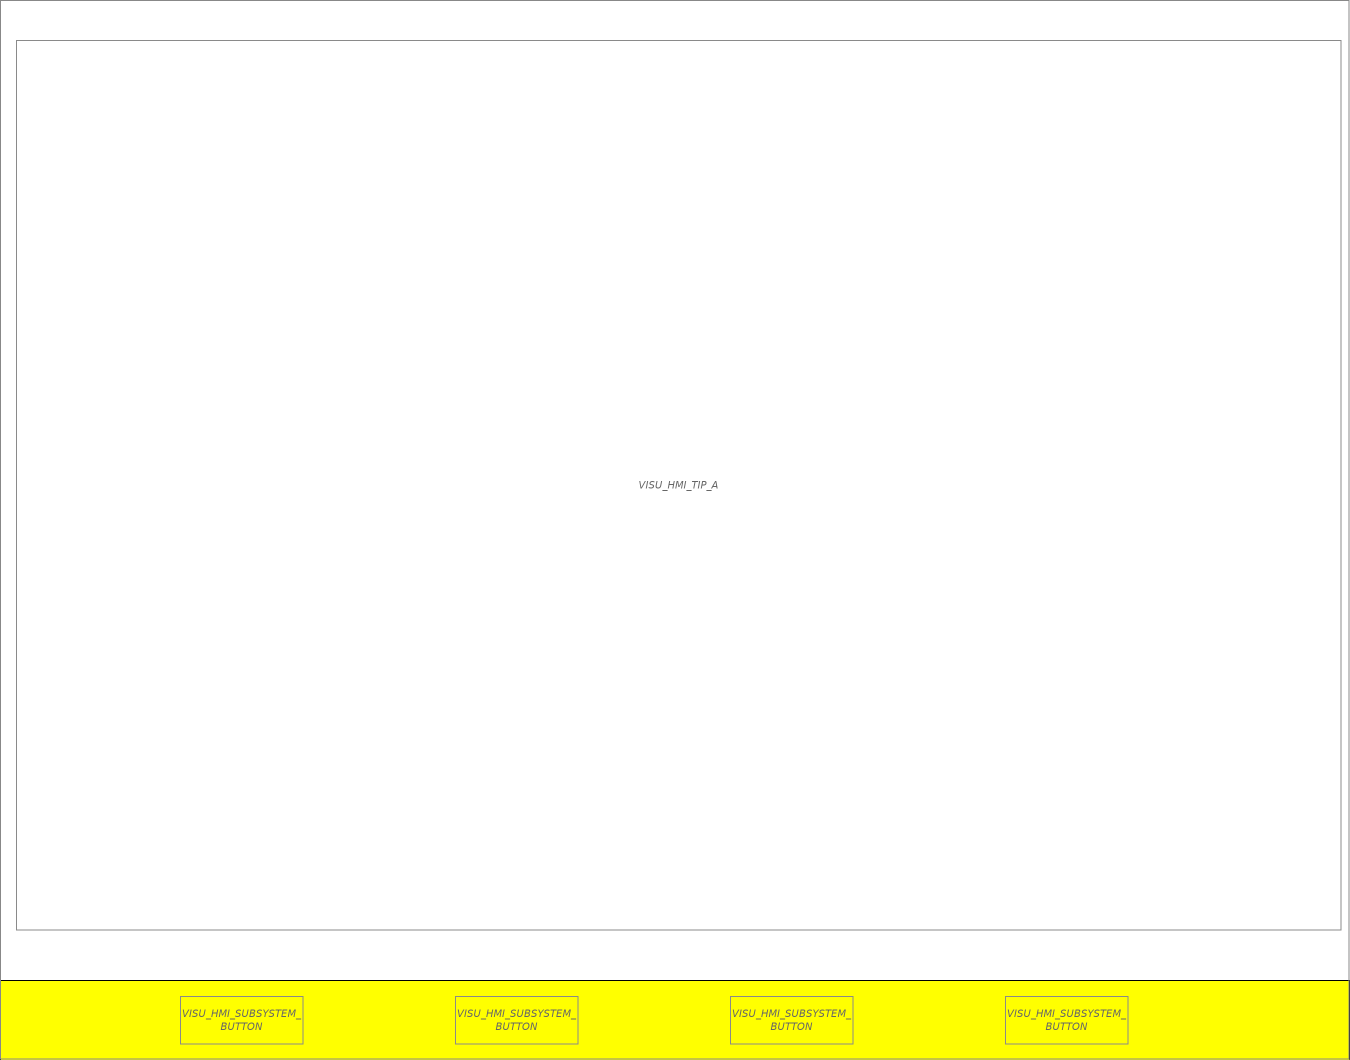
VISUALIZATION VISU_HMI_TIP_TILT  // 1350x1060
VAR_IN_OUT
	m_Hmi : FB_HMI_TIP_TILT;
END_VAR
    Label (10,10 199x30), "Tip Tilt"
    Rectangle (0,980 1350x81)
    Frame (180,996 123x48)
        shows VISU_HMI_SUBSYSTEM_BUTTON(m_Hmi := PRG_HMI.fbTipTilt.fbTipAButton)
        OnMouseClick: execute { m_Hmi.eActiveTab := E_HMI_TIP_TILT_TABS.TIP_A; }
    Frame (455,996 123x48)
        shows VISU_HMI_SUBSYSTEM_BUTTON(m_Hmi := PRG_HMI.fbTipTilt.fbTipBButton)
        OnMouseClick: execute { m_Hmi.eActiveTab := E_HMI_TIP_TILT_TABS.TIP_B; }
    Frame (730,996 123x48)
        shows VISU_HMI_SUBSYSTEM_BUTTON(m_Hmi := PRG_HMI.fbTipTilt.fbTiltAButton)
        OnMouseClick: execute { m_Hmi.eActiveTab := E_HMI_TIP_TILT_TABS.TILT_A; }
    Frame (1005,996 123x48)
        shows VISU_HMI_SUBSYSTEM_BUTTON(m_Hmi := PRG_HMI.fbTipTilt.fbTiltBButton)
        OnMouseClick: execute { m_Hmi.eActiveTab := E_HMI_TIP_TILT_TABS.TILT_B; }
    Frame (16,40 1325x890), frame switch variable: m_Hmi.eActiveTab
        shows VISU_HMI_TIP_A()
        shows VISU_HMI_TIP_B()
        shows VISU_HMI_TILT_A()
        shows VISU_HMI_TILT_B()
END_VISUALIZATION

(* stored: Version 1.1.0.1, ProductVersion 3.1.4024.14
   Visu VISU_HMI_TIP_TILT: Id {40c4923b-bba0-46c7-98e3-8f5f3cae34f2} *)
